FUNCTION_BLOCK PUBLIC FB_ItalianPizzaMozzarella EXTENDS FB_ItalianPizzaMargherita
VAR_INPUT
END_VAR
VAR_OUTPUT
END_VAR
VAR
	bBasil		: BOOL := TRUE;
END_VAR

PROPERTY PUBLIC bHasBasil : BOOL
GET
bHasBasil := this^.bBasil;
END_GET
SET
this^.bBasil := bHasBasil;
END_SET
END_PROPERTY

METHOD PUBLIC GetPrice : LREAL
GetPrice := SUPER^.GetPrice();
IF (THIS^.bBasil) THEN
	GetPrice := GetPrice + 0.25;
END_IF
END_METHOD

END_FUNCTION_BLOCK

(* stored: Version 1.1.0.1, ProductVersion 3.1.4022.16
   POU FB_ItalianPizzaMozzarella: Id {ea223156-5b5e-4799-9284-792e4c0e2e89}, SpecialFunc None
   Property bHasBasil: Id {290a5c31-2e4f-456e-919d-ac60c6ffd80e}
   Get Get: Id {f31e073b-9fb7-474c-9662-43d551eda861}
   Set Set: Id {18c0d77a-acd5-4bb2-ad60-1dc062be8d93}
   Method GetPrice: Id {8906e813-e3da-4856-8d4c-80974f72848b} *)
